PROGRAM MAIN
VAR
	i					: UINT;
	ii					: UINT;
	fbGetCurTaskIndex 	: GETCURTASKINDEX;
	_iDataPos 			: INT;
	_dDataOff 			: DINT;	
	
	LasitManager : FB_LasitManager;
	Lasit 		: FB_Lasit;
	LasitFlyPowerMarkManager : FB_FlyPowerMarkManager;
	St04_MarkingData : DUT_stMarkingData;
	
	fbFlyPowerMarkExeManager : FB_FlyPowerMarkExeManager;
	fbFlyPowerMarkExeManagerInit : BOOL;

// ShiftData	
	stTempData  		: stShiftData;
	//fbShiftManData 		: FB_PartDataManager;
	fbShiftDataBuffer 	: FB_DataBufferManager;
	RTRIG_ShiftTrigger 	: R_TRIG;
	ShiftData 			: ARRAY[0..20] OF stShiftData;
	
	OvrMultiplierOld	: USINT;
	TON_OvrMultFeedback : TON;
	
	_j		  : DINT;
	fbDataRequest		: FB_DataRequest;
	RTRIG_ExecuteWriteChip : R_TRIG;
	RTRIG_ExecuteReadChip : R_TRIG;
	
	tempString1 : STRING;
	tempString2 : STRING;
	tempLayout  : STRING;

	sSrvNetID		: T_AmsNetID	:= '';(* TwinCAT TCP/IP server network address *)
	bEnable			: BOOL 			:= FALSE;(* TRUE => Enable client data exchange, FALSE => Disable *)
	bLog			: BOOL			:= FALSE;(* TRUE => Enable log message output, FALSE => Disable *)

	fbCloseAll		: FB_SocketCloseAll;
	bInitialize		: BOOL := TRUE;
	OvrMng			: FB_OvrMng;
	
	tempString	: STRING;
	tempStringPos : INT;
	
	
	tempPPString			: STRING;
	iPP						: INT;
	
	RTRIG_ProcessingDataExecute	 : R_TRIG;
	RTRIG_ProcessingDataDoneError	: R_TRIG;
	
	tTimeTemp					: TIME := T#100ms;
	TempInt						: UINT;
	tempCouth					: BOOL;
	
	RTRIG_GoodPieces			: R_TRIG;
	RTRIG_Scraped				: R_TRIG;
	RTRIG_BatchChange			: R_TRIG;
	TepmStatus					: eProductStatus;	
	
	RTRIG_UnloadFromSlide		: R_TRIG;
	RTRIG_UnloadFromLaser		: R_TRIG;
	RTRIG_UnloadFromCart		: R_TRIG;
	RTRIG_UnloadFromDeburring	: R_TRIG;
	RTRIG_UnloadFromPallet		: R_TRIG;	
	RTRIG_UnloadFromManualLoad	: R_TRIG;	
	RTRIG_IdShift		: R_TRIG;
	
	RTRIG_UnloadFromSlideAck		: R_TRIG;
	RTRIG_UnloadFromLaserAck		: R_TRIG;
	RTRIG_UnloadFromCartAck			: R_TRIG;
	RTRIG_UnloadFromDeburringAck	: R_TRIG;
	RTRIG_UnloadFromPalletAck		: R_TRIG;
	RTRIG_UnloadFromManualLoadAck	: R_TRIG;
	
	FTRIG_UnloadFromSlideAck		: F_TRIG;
	FTRIG_UnloadFromLaserAck		: F_TRIG;
	FTRIG_UnloadFromCartAck			: F_TRIG;
	FTRIG_UnloadFromDeburringAck	: F_TRIG;
	FTRIG_UnloadFromPalletAck		: F_TRIG;
	FTRIG_UnloadFromManualLoadAck	: F_TRIG;
	
	CycleTime					: DWORD;
	ProcessingHMIDataManager : FB_ButtonTrigger;
	
	fbLoadingModeSelection: FB_LoadingModeChange; 
	
	manualReq : BOOL;
	LasitManualDisable : BOOL;
	fbKillMultipleNavigationPS : FB_KillMultipleNavigationPS;
	tempDint	: ARRAY[0..3] OF DINT;
	tempReal	: ARRAY[0..3] OF REAL;
	resetManual : BOOL;
	RobotLoadOffset : ARRAY[0..EC.NUM_ROBOT_OFFSET - 1] OF DUT_XYZ_Int;
	RobotUnloadOffset : ARRAY[0..EC.NUM_ROBOT_OFFSET - 1] OF DUT_XYZ_Int;
	TON_MSSQL_UpdatePartLocationsAndProcessingDataBusy : TON;
	memReq : BOOL;
	RTRIG_MSSQL_spGetProcessingDataForHMIDone : R_TRIG;
	RTRIG_MSSQL_spGetProcessingDataForHMIExecute : R_TRIG;
	IdList	: ARRAY[0..10] OF DINT;
END_VAR

fbGetCurTaskIndex();

A_00_Init();			// Initialization

/////////INPUT//////////////////////////////////////////////////////////
A_10_EC_PN_Input();				// Profinet to Ethercat
A_11_MatManager_Input();		// Buttons-Leds exchange data	

////////////////////////////////////////////////////////////////////////
//Database();

//A_30_Laser();
A_70_DataRequest();
A_80_OvrMng();

fbLoadingModeSelection(ActualMode := G.LoadingModeActive,
					  	LoadingModeSelected:= HMI.SelectedLoadingMode,
						LS_AutoMode := HMI.General.Manuals.LS[58],
						LS_ManualMode := HMI.General.Manuals.LS[56],
						LS_SemiAutoMode:= HMI.General.Manuals.LS[57],
						PS_AutoMode => HMI.General.Manuals.PS[58],
						PS_ManualMode => HMI.General.Manuals.PS[56],
						PS_SemiAutoMode => HMI.General.Manuals.PS[57]);

PRG_Diagnostic();

/////////OUTPUT//////////////////////////////////////////////////////////
A_90_EC_PN_Output();			// Profinet to Ethercat
A_91_MatManager_Output();			// Buttons-Leds exchange data

////////////////////////////////////////////////////////////////////////

ACTION A_00_Init:
IF _TaskInfo[fbGetCurTaskIndex.index].FirstCycle THEN	// First cycle of this task
	G.Ovr_CounterValue := EC.I_Ovr_CounterValue;
	
	//PRG_MSSQL_InitConnection.Enable := TRUE;
	DB.MesReadStatusCmd := TRUE;
	
	LasitManager.Init := TRUE;
	//fbFlyPowerMarkExeManagerInit := TRUE;
ELSE
	LasitManager.Init := FALSE;
END_IF
END_ACTION

ACTION A_10_EC_PN_Input:
// EV
AL671[0] := I_Y400[0];
AL671[1] := I_Y400[1];
AL671[2] := I_Y400[2];
AL671[3] := I_Y400[3];
AL671[4] := I_Y400[4];
            
AL673[0] := I_Y400[5];
AL673[1] := I_Y400[6];
AL673[2] := I_Y400[7];
AL673[3] := I_Y400[8];
AL673[4] := I_Y400[9];
AL673[5] := I_Y400[10];

////////////////////////////////////////////////////////// Memorie R

HMI.Out.KebaEnabled := I_R2200[0].0;
G.ResetButton := CNC.vKeyboard.PS[16] OR I_R2200[0].1 OR resetManual;

//ShiftData
PRG_MSSQL_spCMD_AbortProduction.Execute 	:= I_R2200[20].2;

//// Laser
LasitManager.Execute := I_R2200[25].0 OR manualReq;
G.LasitOn			:= I_R2200[25].1;


G.MachineEmpty					:= I_R2200[40].0;
HMI.out.EnableProductionAction 	:= I_R2200[41].1;

RTRIG_UnloadFromSlide.CLK := I_R2200[42].0;
RTRIG_UnloadFromLaser.CLK := I_R2200[42].1;
RTRIG_UnloadFromCart.CLK := I_R2200[42].2;
RTRIG_UnloadFromDeburring.CLK := I_R2200[42].3;
RTRIG_UnloadFromPallet.CLK := I_R2200[42].4;
RTRIG_UnloadFromManualLoad.CLK := I_R2200[42].5;
////////////////////////////////////////////////////////// Memorie D

// WId macchina e stato pezzo
FOR _iDataPos := 1 TO CNC.NUM_DATA_POSITION+3 DO
	_dDataOff := (_iDataPos)*5;	
	MEMCPY(ADR(HMI.ShiftData[_iDataPos].FLAGP.aByte), ADR(CNC.I_D2200[_dDataOff]), SIZEOF(BYTE));
	MEMCPY(ADR(HMI.ShiftData[_iDataPos].WIDP), ADR(CNC.I_D2200[_dDataOff+1]), SIZEOF(DWORD));
END_FOR

// feedback pennetta
MEMCPY(ADR(tempDint[0]), ADR(CNC.I_D2200[100]), SIZEOF(DWORD));
tempReal[0] := TO_REAL(tempDint[0]);
HMI.Out.Probe.ActualEncoderValue := tempReal[0]/1000;

MEMCPY(ADR(tempDint[1]), ADR(CNC.I_D2200[104]), SIZEOF(DWORD));
tempReal[1] := TO_REAL(tempDint[1]);
HMI.Out.Probe.ActualProbeValue := tempReal[1]/1000;
HMI.Out.Probe.Error := CNC.I_D2200[108].0;
END_ACTION

ACTION A_11_MatManager_Input:
FC_BYTE_TO_BOOLARR(ADR(HMI.General.Manuals.LS), ADR(CNC.I_R4500[0]), SIZEOF(HMI.General.Manuals.LS));
FC_BYTE_TO_BOOLARR(ADR(HMI.St0.Manuals.LS), ADR(CNC.I_R4500[60]), SIZEOF(HMI.St0.Manuals.LS));
FC_BYTE_TO_BOOLARR(ADR(HMI.St1.Manuals.LS), ADR(CNC.I_R4500[100]), SIZEOF(HMI.St1.Manuals.LS));
FC_BYTE_TO_BOOLARR(ADR(HMI.St2.Manuals.LS), ADR(CNC.I_R4500[110]), SIZEOF(HMI.St2.Manuals.LS));
FC_BYTE_TO_BOOLARR(ADR(HMI.St3.Manuals.LS), ADR(CNC.I_R4500[120]), SIZEOF(HMI.St3.Manuals.LS));
FC_BYTE_TO_BOOLARR(ADR(HMI.St4.Manuals.LS), ADR(CNC.I_R4500[130]), SIZEOF(HMI.St4.Manuals.LS));
FC_BYTE_TO_BOOLARR(ADR(HMI.St5.Manuals.LS), ADR(CNC.I_R4500[140]), SIZEOF(HMI.St5.Manuals.LS));
FC_BYTE_TO_BOOLARR(ADR(HMI.St6.Manuals.LS), ADR(CNC.I_R4500[150]), SIZEOF(HMI.St6.Manuals.LS));
FC_BYTE_TO_BOOLARR(ADR(HMI.St7.Manuals.LS), ADR(CNC.I_R4500[160]), SIZEOF(HMI.St7.Manuals.LS));
FC_BYTE_TO_BOOLARR(ADR(HMI.St8.Manuals.LS), ADR(CNC.I_R4500[170]), SIZEOF(HMI.St8.Manuals.LS));
FC_BYTE_TO_BOOLARR(ADR(HMI.St9.Manuals.LS), ADR(CNC.I_R4500[180]), SIZEOF(HMI.St9.Manuals.LS));
FC_BYTE_TO_BOOLARR(ADR(HMI.St10.Manuals.LS), ADR(CNC.I_R4500[190]),	SIZEOF(HMI.St10.Manuals.LS));
FC_BYTE_TO_BOOLARR(ADR(HMI.St11.Manuals.LS), ADR(CNC.I_R4500[200]),	SIZEOF(HMI.St11.Manuals.LS));
FC_BYTE_TO_BOOLARR(ADR(HMI.St12.Manuals.LS), ADR(CNC.I_R4500[210]),	SIZEOF(HMI.St12.Manuals.LS));
FC_BYTE_TO_BOOLARR(ADR(HMI.St13.Manuals.LS), ADR(CNC.I_R4500[220]),	SIZEOF(HMI.St13.Manuals.LS));

//Navigation
FC_BYTE_TO_BOOLARR(ADR(HMI.In.Navigation.LS[0]), ADR(CNC.I_R4500[350]), HMI.NUM_NAVIGATION_ITEMS);

// vKeyboard
FC_BYTE_TO_BOOLARR(ADR(CNC.vKeyboard.LS), ADR(CNC.I_R3950), SIZEOF(CNC.vKeyboard.LS));

//MachineData Header
FC_BYTE_TO_BOOLARR(ADR(MachineData.aBool), ADR(CNC.I_E0000[0]), SIZEOF(MachineData.aBool));
MEMCPY(ADR(MachineData.aByte), ADR(CNC.I_E0000[10]), SIZEOF(MachineData.aByte));
MEMCPY(ADR(MachineData.aWord), ADR(CNC.I_E0000[20]), SIZEOF(MachineData.aWord));

//Safety
MEMCPY(ADR(HMI.Out.Gc1000Status), ADR(CNC.I_E0000[29]), SIZEOF(HMI.Out.Gc1000Status));
MEMCPY(ADR(HMI.Out.Doors), ADR(CNC.I_E0000[30]), SIZEOF(HMI.Out.Doors));

//Counters
MEMCPY(ADR(HMI.Out.Counters.TotalPieceGood), ADR(CNC.I_E0000[60]), SIZEOF(DWORD));
MEMCPY(ADR(HMI.Out.Counters.TotalPieceScrap), ADR(CNC.I_E0000[64]), SIZEOF(DWORD));
	
// Machine CycleTime
MEMCPY(ADR(CycleTime), ADR(CNC.I_E0000[96]), SIZEOF(CycleTime));
	
//MachineData Station	
MEMCPY(ADR(MachineData.aSt[1]), ADR(CNC.I_E0000[100]), SIZEOF(MachineData.aSt));

// Lasit - senza indirizzo MB
LasitFlyPowerMarkManager.In := (CNC.FlyPowerMarkOn = 1);	

//Richiesta dato
MEMCPY(ADR(DataRequestRead.aByte[0]), ADR(CNC.HS_read[0]), SIZEOF(BYTE));
MEMCPY(ADR(DataRequestRead.aDWord), ADR(CNC.HS_read[6]), SIZEOF(DWORD));
END_ACTION

ACTION A_30_Laser:
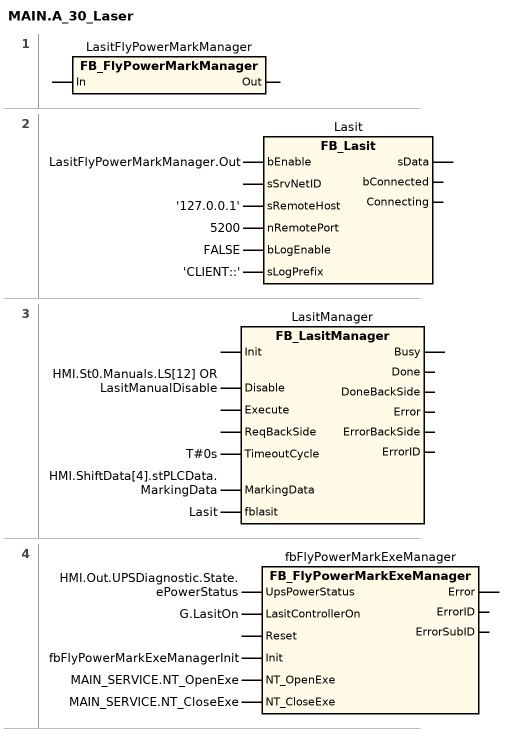
// NETWORK 1
LasitFlyPowerMarkManager(); // FB_FlyPowerMarkManager

// NETWORK 2
Lasit(
    bEnable := LasitFlyPowerMarkManager.Out,
    sRemoteHost := '127.0.0.1',
    nRemotePort := 5200,
    bLogEnable := FALSE,
    sLogPrefix := 'CLIENT::'); // FB_Lasit

// NETWORK 3
LasitManager(
    Disable := HMI.St0.Manuals.LS[12] OR LasitManualDisable,
    TimeoutCycle := T#0s,
    MarkingData := HMI.ShiftData[4].stPLCData.MarkingData,
    fblasit := Lasit); // FB_LasitManager

// NETWORK 4
fbFlyPowerMarkExeManager(
    UpsPowerStatus := HMI.Out.UPSDiagnostic.State.ePowerStatus,
    LasitControllerOn := G.LasitOn,
    Init := fbFlyPowerMarkExeManagerInit,
    NT_OpenExe := MAIN_SERVICE.NT_OpenExe,
    NT_CloseExe := MAIN_SERVICE.NT_CloseExe); // FB_FlyPowerMarkExeManager
END_ACTION

ACTION A_70_DataRequest:
fbDataRequest( ExecuteCurrent  := CNC.DataRequestRead.aByte[0].aBit.b0 OR G.RequestActual,
			   ExecuteNext	:= CNC.DataRequestRead.aByte[0].aBit.b1 OR G.RequestNext, 
			   Reset 		:= G.ResetButton,
			   WID			:= CNC.DataRequestRead.aDWord,
			   WID_Old		:= G.WID_Old,
			   MachineEmpty	:= G.MachineEmpty,
			   Done			=> CNC.DataRequestWrite.aByte[0].aBit.b0,
			   Busy			=> ,
			   Error		=> CNC.DataRequestWrite.aByte[0].aBit.b1,
			   ErrorCodePMC => CNC.DataRequestWrite.aByte[1].aByte,		 
			   St0Data 		:= St0DataTemp,
			   PMC_ShiftManData0 := HMI.ShiftData[0],
			   fbShiftDataBuffer := fbShiftDataBuffer);
			   
fbShiftDataBuffer(ArraySize := UINT_TO_INT(G.DATABUFFER_SIZE), DataRepository := ADR(G.DataBuffer));
FOR i := 1 TO NUM_STATIONS DO
	FC_DataFind(HMI.ShiftData[i].WIDP, ADR(HMI.ShiftData[i].PmcData), ADR(HMI.ShiftData[i].stPLCData), ADR(G.DataBuffer));
	IF HMI.ShiftData[i].WIDP = DB.ProcessingHMIDataLocation[i].PartId THEN	
		HMI.ShiftData[i].ProcessingData := DB.ProcessingHMIDataViewData[i];
	END_IF
END_FOR

FOR i := 0 TO NUM_STATIONS DO
	IdList[i] := HMI.ShiftData[i].WIDP;
END_FOR

IF NOT G.MachineEmpty AND MEMCMP(ADR(IdList), ADR(G.IdList_Old), SIZEOF(IdList)) <> 0 THEN
	G.UpdatePartLocationsAndProcessingDataTrigger := TRUE;
	MEMCPY(ADR(G.IdList_Old), ADR(IdList), SIZEOF(G.IdList_Old));
END_IF

//unload managment
//////////////////////Prima di rimuovere i dati dalla struttura mi salvo info per gestire tutto il resto //////////////////////
////////////////////// updateProcessingData per database, dati per oee per sapere se pezzo ok o scarto //////////////////////
////////////////////// NOTA LA POSIZIONE 17 è DOVE VENGONO SALVATI I DATI DEL PEZZO SCARICATO DAL PMC //////////////////////

IF RTRIG_UnloadFromSlide.Q THEN
	FC_UnloadManager(G.fbProcessingData[1].UnloadingStation, HMI.ShiftData[17].FLAGP);
	G.PMCShiftDataSlide := HMI.ShiftData[17];
	FC_OeeSetUpdateCount(HMI.ShiftData[17].FLAGP);
	FC_UpdatePieceCount(HMI.ShiftData[17].FLAGP, ADR(HMI.Out.Header.Pieces));
END_IF
IF RTRIG_UnloadFromLaser.Q THEN
	FC_UnloadManager(G.fbProcessingData[2].UnloadingStation, HMI.ShiftData[17].FLAGP);
	G.PMCShiftDataLaser := HMI.ShiftData[17];
	FC_OeeSetUpdateCount(HMI.ShiftData[17].FLAGP);
	FC_UpdatePieceCount(HMI.ShiftData[17].FLAGP, ADR(HMI.Out.Header.Pieces));
END_IF
IF RTRIG_UnloadFromCart.Q THEN
	FC_UnloadManager(G.fbProcessingData[5].UnloadingStation, HMI.ShiftData[17].FLAGP);
	G.PMCShiftDataCart := HMI.ShiftData[17];
	FC_OeeSetUpdateCount(HMI.ShiftData[17].FLAGP);
	FC_UpdatePieceCount(HMI.ShiftData[17].FLAGP, ADR(HMI.Out.Header.Pieces));
END_IF
IF RTRIG_UnloadFromDeburring.Q THEN
	FC_UnloadManager(G.fbProcessingData[8].UnloadingStation, HMI.ShiftData[17].FLAGP);
	G.PMCShiftDataDeburring := HMI.ShiftData[17];
	FC_OeeSetUpdateCount(HMI.ShiftData[17].FLAGP);
	FC_UpdatePieceCount(HMI.ShiftData[17].FLAGP, ADR(HMI.Out.Header.Pieces));
END_IF
IF RTRIG_UnloadFromPallet.Q THEN
	FC_UnloadManager(G.fbProcessingData[9].UnloadingStation, HMI.ShiftData[17].FLAGP);
	G.PMCShiftDataPallet := HMI.ShiftData[17];
	FC_OeeSetUpdateCount(HMI.ShiftData[17].FLAGP);
	FC_UpdatePieceCount(HMI.ShiftData[17].FLAGP, ADR(HMI.Out.Header.Pieces));
END_IF
IF RTRIG_UnloadFromManualLoad.Q THEN
	FC_UnloadManager(G.fbProcessingData[14].UnloadingStation, HMI.ShiftData[17].FLAGP);
	G.PMCShiftDataPallet := HMI.ShiftData[17];
	FC_OeeSetUpdateCount(HMI.ShiftData[17].FLAGP);
	FC_UpdatePieceCount(HMI.ShiftData[17].FLAGP, ADR(HMI.Out.Header.Pieces));	
END_IF

RTRIG_UnloadFromSlide(Q => DB.fbTriggerSequencer.In[0]);
RTRIG_UnloadFromLaser(Q => DB.fbTriggerSequencer.In[1]);
RTRIG_UnloadFromCart(Q => DB.fbTriggerSequencer.In[2]);
RTRIG_UnloadFromDeburring(Q => DB.fbTriggerSequencer.In[3]);
RTRIG_UnloadFromPallet(Q => DB.fbTriggerSequencer.In[4]);
RTRIG_UnloadFromManualLoad(Q => DB.fbTriggerSequencer.In[5]);
RTRIG_IdShift(CLK := G.UpdatePartLocationsAndProcessingDataTrigger,Q => DB.fbTriggerSequencer.In[5]);

//////////////////////////////////////////////////////////////////////////////
// dopo UpdatePartLocationAndProcessingData posso richiedere a database i ProcessingDataHMI aggiornati 	   
//RTRIG_ProcessingHMIDataExecute(CLK:= PRG_MSSQL_UpdatePartLocationsAndProcessingData.Done);
TON_MSSQL_UpdatePartLocationsAndProcessingDataBusy(IN := NOT PRG_MSSQL_UpdatePartLocationsAndProcessingData.Busy AND NOT PRG_MSSQL_UpdatePartLocationsAndProcessingData.Execute, PT := T#100MS);
ProcessingHMIDataManager(I_Command			:= (fbDataRequest.Done OR PRG_MSSQL_UpdatePartLocationsAndProcessingData.Done)
												AND NOT PRG_MSSQL_UpdatePartLocationsAndProcessingData.Execute AND NOT PRG_MSSQL_UpdatePartLocationsAndProcessingData.Busy,
                     	 I_CommandEnable	:= TRUE,	
                     	 I_Reset			:= PRG_MSSQL_spGetProcessingDataForHMI.Done OR PRG_MSSQL_spGetProcessingDataForHMI.Error,	
                     	 I_ResetEnable		:= TRUE,
						 Q_Out				:= PRG_MSSQL_spGetProcessingDataForHMI.Execute);

RTRIG_MSSQL_spGetProcessingDataForHMIDone(CLK := PRG_MSSQL_spGetProcessingDataForHMI.Done);						 
IF RTRIG_MSSQL_spGetProcessingDataForHMIDone.Q THEN
	memReq := TRUE;
END_IF

IF memReq AND NOT HMI.Out.ProductionQueueRefresh THEN
	memReq := FALSE;
END_IF
END_ACTION

ACTION A_80_OvrMng:

IF MachineData.aByte[3] <> 10 AND MachineData.aByte[3] <> 1 THEN
	OvrMng.I_Multiplier := 1;
ELSE
	OvrMng.I_Multiplier := MachineData.aByte[3];
END_IF


OvrMng(
	I_CounterValue 		:= EC.I_Ovr_CounterValue,
	I_SetCounterDone 	:= EC.I_Ovr_SetCounterDone,
	I_Overflow			:= EC.I_Ovr_Overflow,
	I_Underflow			:= EC.I_Ovr_Underflow,
	I_CounterValueOld	:= G.Ovr_CounterValue,
	I_Multiplier		:=,
	I_SetCounter		:=,
	I_SetCounterValue	:=,
	I_OvrMaxValue		:= 100,
	I_OvrMinValue		:= 0,
	Q_SetCounter 		=> EC.Q_Ovr_SetCounter,
	Q_SetCounterValue	=> EC.Q_Ovr_SetCounterValue,
	Q_Ovr				:= G.Ovr
);
END_ACTION

ACTION A_90_EC_PN_Output:
////////////////////////////////////////////////////////// Memorie R
/// allarme beckhoff ferma in fase PMC
Q_R2000[0].0 := MAIN_SERVICE.MSSQL_Events.Cumulative OR MAIN_SERVICE.Marker_Events.Cumulative OR MAIN_SERVICE.DataRequest_Events.Cumulative;

//Svuotamento forzato
CNC.Q_R2000[20].2 := PRG_MSSQL_spCMD_AbortProduction.Done;
CNC.Q_R2000[20].3 := PRG_MSSQL_spCMD_AbortProduction.Error;

//// Laser
Q_R2000[25].0 := LasitManager.Done;	
Q_R2000[25].1 := LasitManager.Error;

// Ack unload trigger
RTRIG_UnloadFromSlideAck(CLK := G.fbProcessingData[1].UnloadingStation);
RTRIG_UnloadFromLaserAck(CLK := G.fbProcessingData[2].UnloadingStation);
RTRIG_UnloadFromCartAck(CLK := G.fbProcessingData[5].UnloadingStation);
RTRIG_UnloadFromDeburringAck(CLK := G.fbProcessingData[8].UnloadingStation);
RTRIG_UnloadFromPalletAck(CLK := G.fbProcessingData[9].UnloadingStation);
RTRIG_UnloadFromManualLoadAck(CLK := G.fbProcessingData[14].UnloadingStation);

FTRIG_UnloadFromSlideAck(CLK := RTRIG_UnloadFromSlide.CLK);
FTRIG_UnloadFromLaserAck(CLK := RTRIG_UnloadFromLaser.CLK);
FTRIG_UnloadFromCartAck(CLK := RTRIG_UnloadFromCart.CLK);
FTRIG_UnloadFromDeburringAck(CLK := RTRIG_UnloadFromDeburring.CLK);
FTRIG_UnloadFromPalletAck(CLK := RTRIG_UnloadFromPallet.CLK);
FTRIG_UnloadFromManualLoadAck(CLK := RTRIG_UnloadFromManualLoad.CLK);

IF RTRIG_UnloadFromSlideAck.Q THEN 		Q_R2000[42].0 := TRUE; END_IF
IF RTRIG_UnloadFromLaserAck.Q THEN 		Q_R2000[42].1 := TRUE; END_IF
IF RTRIG_UnloadFromCartAck.Q THEN 		Q_R2000[42].2 := TRUE; END_IF
IF RTRIG_UnloadFromDeburringAck.Q THEN 	Q_R2000[42].3 := TRUE; END_IF
IF RTRIG_UnloadFromPalletAck.Q THEN 	Q_R2000[42].4 := TRUE; END_IF
IF RTRIG_UnloadFromManualLoadAck.Q THEN 	Q_R2000[42].5 := TRUE; END_IF

IF FTRIG_UnloadFromSlideAck.Q THEN 		Q_R2000[42].0 := FALSE; END_IF
IF FTRIG_UnloadFromLaserAck.Q THEN 		Q_R2000[42].1 := FALSE; END_IF
IF FTRIG_UnloadFromCartAck.Q THEN 		Q_R2000[42].2 := FALSE; END_IF
IF FTRIG_UnloadFromDeburringAck.Q THEN 	Q_R2000[42].3 := FALSE; END_IF
IF FTRIG_UnloadFromPalletAck.Q THEN 	Q_R2000[42].4 := FALSE; END_IF
IF FTRIG_UnloadFromManualLoadAck.Q THEN 	Q_R2000[42].5 := FALSE; END_IF

////////////////////////////////////////////////////////// Memorie D

//Ovr
CNC.Q_D2000[0] := G.Ovr;

//Robot load override 
CNC.Q_D2000[2] := TO_BYTE( MIN(HMI.RobotLoadSetpoint.Override, EC.NUM_MAX_ROBOT_OVR) );

//Robot unload override 
CNC.Q_D2000[3] := TO_BYTE( MIN(HMI.RobotUnloadSetpoint.Override, EC.NUM_MAX_ROBOT_OVR) );

// soglie pennetta
HMI.Out.Probe.UpperLimit := 0.1;
tempDint[2] := TO_DINT(HMI.Out.Probe.UpperLimit*1000);
MEMCPY(ADR(CNC.Q_D2000[4]), ADR(tempDint[2]), SIZEOF(DWORD));
HMI.Out.Probe.LowerLimit := -0.1;
tempDint[3] := TO_DINT(HMI.Out.Probe.LowerLimit*1000);
MEMCPY(ADR(CNC.Q_D2000[8]), ADR(tempDint[3]), SIZEOF(DWORD));

// questo serve perchè pannello fa schifo
IF HMI.St4.BroachTarget = 0 THEN HMI.St4.BroachTarget := 1; END_IF
IF HMI.St5.BroachTarget = 0 THEN HMI.St5.BroachTarget := 1; END_IF
IF HMI.St6.BroachTarget = 0 THEN HMI.St6.BroachTarget := 1; END_IF
IF HMI.St7.BroachTarget = 0 THEN HMI.St7.BroachTarget := 1; END_IF
IF HMI.St8.BroachTarget = 0 THEN HMI.St8.BroachTarget := 1; END_IF
IF HMI.St9.BroachTarget = 0 THEN HMI.St9.BroachTarget := 1; END_IF
IF HMI.St10.BroachTarget = 0 THEN HMI.St10.BroachTarget := 1; END_IF

// Broccia tagert per comando vai a
CNC.Q_D2000[20] := TO_BYTE( MAX( MIN(HMI.St4.BroachTarget,  EC.NUM_MAX_BROACH), EC.NUM_MIN_BROACH) );
CNC.Q_D2000[21] := TO_BYTE( MAX( MIN(HMI.St5.BroachTarget,  EC.NUM_MAX_BROACH), EC.NUM_MIN_BROACH) );
CNC.Q_D2000[22] := TO_BYTE( MAX( MIN(HMI.St6.BroachTarget,  EC.NUM_MAX_BROACH), EC.NUM_MIN_BROACH) );
CNC.Q_D2000[23] := TO_BYTE( MAX( MIN(HMI.St7.BroachTarget,  EC.NUM_MAX_BROACH), EC.NUM_MIN_BROACH) );
CNC.Q_D2000[24] := TO_BYTE( MAX( MIN(HMI.St8.BroachTarget,  EC.NUM_MAX_BROACH), EC.NUM_MIN_BROACH) );
CNC.Q_D2000[25] := TO_BYTE( MAX( MIN(HMI.St9.BroachTarget,  EC.NUM_MAX_BROACH), EC.NUM_MIN_BROACH) );
CNC.Q_D2000[26] := TO_BYTE( MAX( MIN(HMI.St10.BroachTarget, EC.NUM_MAX_BROACH), EC.NUM_MIN_BROACH) );

// dragante
MEMCPY(ADR(CNC.Q_D2000[28]), ADR(HMI.ChipConveyorSetpoint), SIZEOF(WORD));

// dragante
MEMCPY(ADR(CNC.Q_D2000[30]), ADR(HMI.DropsaSetpoint), SIZEOF(WORD));

//Robot load offset
FOR i := 0 TO EC.NUM_ROBOT_OFFSET - 1 DO
	RobotLoadOffset[i].X := TO_INT(HMI.RobotLoadSetpoint.PositionOffset[i].X *1000);
	RobotLoadOffset[i].Y := TO_INT(HMI.RobotLoadSetpoint.PositionOffset[i].Y *1000);
	RobotLoadOffset[i].Z := TO_INT(HMI.RobotLoadSetpoint.PositionOffset[i].Z *1000);
END_FOR
MEMCPY(ADR(CNC.Q_D2000[40]), ADR(RobotLoadOffset), SIZEOF(DUT_XYZ_Int)*EC.NUM_ROBOT_OFFSET);

//Robot unload offset
FOR i := 0 TO EC.NUM_ROBOT_OFFSET - 1 DO
	RobotUnloadOffset[i].X := TO_INT(HMI.RobotUnloadSetpoint.PositionOffset[i].X *1000);
	RobotUnloadOffset[i].Y := TO_INT(HMI.RobotUnloadSetpoint.PositionOffset[i].Y *1000);
	RobotUnloadOffset[i].Z := TO_INT(HMI.RobotUnloadSetpoint.PositionOffset[i].Z *1000);
END_FOR	
MEMCPY(ADR(CNC.Q_D2000[64]), ADR(RobotUnloadOffset), SIZEOF(DUT_XYZ_Int)*EC.NUM_ROBOT_OFFSET);
END_ACTION

ACTION A_91_MatManager_Output:
FC_BOOLARR_TO_BYTE(ADR(CNC.Q_R4000[0]), ADR(HMI.General.Manuals.PS), SIZEOF(HMI.General.Manuals.PS));
FC_BOOLARR_TO_BYTE(ADR(CNC.Q_R4000[60]), ADR(HMI.St0.Manuals.PS), SIZEOF(HMI.St0.Manuals.PS));
FC_BOOLARR_TO_BYTE(ADR(CNC.Q_R4000[100]), ADR(HMI.St1.Manuals.PS), SIZEOF(HMI.St1.Manuals.PS));
FC_BOOLARR_TO_BYTE(ADR(CNC.Q_R4000[110]), ADR(HMI.St2.Manuals.PS), SIZEOF(HMI.St2.Manuals.PS));
FC_BOOLARR_TO_BYTE(ADR(CNC.Q_R4000[120]), ADR(HMI.St3.Manuals.PS), SIZEOF(HMI.St3.Manuals.PS));
FC_BOOLARR_TO_BYTE(ADR(CNC.Q_R4000[130]), ADR(HMI.St4.Manuals.PS), SIZEOF(HMI.St4.Manuals.PS));
FC_BOOLARR_TO_BYTE(ADR(CNC.Q_R4000[140]), ADR(HMI.St5.Manuals.PS), SIZEOF(HMI.St5.Manuals.PS));
FC_BOOLARR_TO_BYTE(ADR(CNC.Q_R4000[150]), ADR(HMI.St6.Manuals.PS), SIZEOF(HMI.St6.Manuals.PS));
FC_BOOLARR_TO_BYTE(ADR(CNC.Q_R4000[160]), ADR(HMI.St7.Manuals.PS), SIZEOF(HMI.St7.Manuals.PS));
FC_BOOLARR_TO_BYTE(ADR(CNC.Q_R4000[170]), ADR(HMI.St8.Manuals.PS), SIZEOF(HMI.St8.Manuals.PS));
FC_BOOLARR_TO_BYTE(ADR(CNC.Q_R4000[180]), ADR(HMI.St9.Manuals.PS), SIZEOF(HMI.St9.Manuals.PS));
FC_BOOLARR_TO_BYTE(ADR(CNC.Q_R4000[190]), ADR(HMI.St10.Manuals.PS), SIZEOF(HMI.St10.Manuals.PS));
FC_BOOLARR_TO_BYTE(ADR(CNC.Q_R4000[200]), ADR(HMI.St11.Manuals.PS), SIZEOF(HMI.St11.Manuals.PS));
FC_BOOLARR_TO_BYTE(ADR(CNC.Q_R4000[210]), ADR(HMI.St12.Manuals.PS), SIZEOF(HMI.St12.Manuals.PS));
FC_BOOLARR_TO_BYTE(ADR(CNC.Q_R4000[220]), ADR(HMI.St13.Manuals.PS), SIZEOF(HMI.St13.Manuals.PS));

//Navigation
// funzione di sicurezza se si inchioda qualcosa a scada per problemi
fbKillMultipleNavigationPS(Ps := ADR(HMI.In.Navigation.PS[0]));
//
FC_BOOLARR_TO_BYTE(ADR(CNC.Q_R4000[350]), ADR(HMI.In.Navigation.PS[0]), HMI.NUM_NAVIGATION_ITEMS);

// vKeyboard
FC_BOOLARR_TO_BYTE(ADR(CNC.Q_R3900), ADR(CNC.vKeyboard.PS), SIZEOF(CNC.vKeyboard.PS));

//Richiesta dato
//MEMCPY(ADR(St0Data), ADR(St0DataTemp), SIZEOF(BYTE)*5);
MEMCPY(ADR(St0Data[0]), ADR(St0DataTemp.FlagP), SIZEOF(BYTE)*6);
MEMCPY(ADR(St0Data[6]), ADR(St0DataTemp.RunP), SIZEOF(DWORD));
MEMCPY(ADR(St0Data[10]), ADR(St0DataTemp.WindP), SIZEOF(DWORD)*2);
MEMCPY(ADR(St0Data[18]), ADR(St0DataTemp.Tpcy), SIZEOF(BYTE)*50);
MEMCPY(ADR(St0Data[68]), ADR(St0DataTemp.Data[1]), SIZEOF(DWORD)*93);
MEMCPY(ADR(St0Data[440]), ADR(St0DataTemp.DataB[1]), SIZEOF(DWORD)*20);
MEMCPY(ADR(St0Data[460]), ADR(St0DataTemp.DataAu[1]), SIZEOF(DWORD)*10);

MEMCPY(ADR(CNC.HS_write[0]), ADR(DataRequestWrite.aByte[0]), SIZEOF(BYTE));
MEMCPY(ADR(CNC.HS_write[1]), ADR(DataRequestWrite.aByte[1]), SIZEOF(BYTE));
MEMCPY(ADR(CNC.HS_write[9]), ADR(DataRequestWrite.aDWord), SIZEOF(DWORD));
END_ACTION

END_PROGRAM

(* stored: Version 1.1.0.1, ProductVersion 3.1.4024.15
   POU MAIN: Id {820a0544-c9ae-49c6-ab68-947b05754ef0}, SpecialFunc None
   Action A_00_Init: Id {c09302aa-9490-43f8-a0bd-7b20dbaacfb4}
   Action A_10_EC_PN_Input: Id {7b76ae9b-1843-4001-b280-19e05c28501a}
   Action A_11_MatManager_Input: Id {79639969-7436-4242-b538-5848cb792d15}
   Action A_30_Laser: Id {998780bc-1d00-4afc-9aa8-e55bab9192fd}
   Action A_70_DataRequest: Id {3461f731-c67f-4176-b757-bd7836528b42}
   Action A_80_OvrMng: Id {d71d79e9-91f9-4f74-addd-612ef513c705}
   Action A_90_EC_PN_Output: Id {3970479d-1672-45b7-8700-f9046a1fe6de}
   Action A_91_MatManager_Output: Id {33101643-ae07-42e3-bbc6-a1fedc00a912} *)
